TYPE ST_ErrorView :
STRUCT
	id:DINT;
	idparam:DINT;
	sMess:STRING[150];
END_STRUCT
END_TYPE

(* stored: Version 1.1.0.1, ProductVersion 3.1.4020.6
   DUT ST_ErrorView: Id {34007b91-303c-4c4f-9766-b6f65829dd8d} *)
